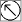
VISUALIZATION VISU_HydraulicsFigure_Manometer  // 22x22
    Ellipse (0,0 20x20)
    Line (5,5) (15,15)
    Line (10,5) (5,5)
    Line (5,10) (5,5)
END_VISUALIZATION

(* stored: Version 1.1.0.1, ProductVersion 3.1.4019.2
   Visu VISU_HydraulicsFigure_Manometer: Id {aefe584f-e8af-4c5f-96a2-86b279ff4afc} *)
